KUKA KRL program: chk_w3_grp2_opn.src

&ACCESS RVP1
&COMMENT Check GRP Z2 ACTROS OPEN
DEF chk_w3_grp2_opn( )

; Check gripper actros OPEN Z2
;//---- Start User-------

$TIMER[10] = 0
$TIMER_STOP[10] = FALSE

WAIT FOR (NOT $IN[10])
WAIT FOR ($IN[9])

$TIMER_STOP[10] = TRUE
$TIMER[10] = 0

;//---- End User---------

END
